{attribute 'monitoring':='call'}
INTERFACE I_CameraSink

METHOD AddCamPoint : BOOL
VAR_INPUT
	sDeformationPoint	: ST_DeformationPointAccurate;
END_VAR
END_METHOD

METHOD AddTeachPoint : BOOL
VAR_INPUT
  sTeachPoint : ST_DeformationPointAccurate;
END_VAR
END_METHOD

END_INTERFACE

(* stored: Version 1.1.0.1, ProductVersion 3.1.4024.3
   Itf I_CameraSink: Id {a2aed62b-000f-44dd-9fef-1bb70d080fae}
   Method AddCamPoint: Id {9b248253-6811-4222-bfe0-383316c5cb83}
   Method AddTeachPoint: Id {9495948b-b7b1-4bb3-8911-32a444e3bfee} *)
